INTERFACE I_StructuredDatatypeAddedEvent EXTENDS I_Event

PROPERTY PUBLIC Target : I_StructuredDatatype
GET
END_GET
END_PROPERTY

END_INTERFACE

(* stored: Version 1.1.0.1, ProductVersion 3.1.4024.12
   Itf I_StructuredDatatypeAddedEvent: Id {6c1ff67b-6aae-02d8-23de-42eb3324db68}
   Property Target: Id {3df22136-2c0b-0878-24c7-5234b92f880e}
   Get Get: Id {24c0a0ed-6d2a-0623-0939-3fa8c2fe089b} *)
